// TIA Portal V15.1 export
// export: Created 2024-06-21T08:40:41.5372667Z, ExportSetting WithDefaults, DisplayName Totally Integrated Automation Portal, DisplayVersion V15.1 Update 5, DisplayName TIA Portal Openness, DisplayVersion V15.1 Update 5, DisplayName SINAMICS Startdrive Advanced, DisplayVersion V15.1, DisplayName G130, G150, S120, S150, SINAMICS MV, S210, DisplayVersion V15.1, DisplayName G110M, G120, G120C, G120D, G120P, DisplayVersion V15.1, DisplayName STEP 7 Professional, DisplayVersion V15.1 Update 5, DisplayName STEP 7 Safety, DisplayVersion V15.1, DisplayName WinCC Professional, DisplayVersion V15.1 Update 5, DisplayName SIMATIC Visualization Architect, DisplayVersion V15.1
DATA_BLOCK "_209000NCP01Passiv"   // DB252
{ S7_Optimized_Access := 'FALSE' }
AUTHOR : VCC
VERSION : 0.1
// stored: AutoNumber false, DBAccessibleFromOPCUA true, IsOnlyStoredInLoadMemory false, IsWriteProtectedInAS false
   VAR RETAIN
      AA_209000AK01JX35IF5010 { ExternalAccessible := 'False'; ExternalVisible := 'False'; ExternalWritable := 'False'} : Bool;   // Passivation alarm - ET200sp I/O - Safety Card IF5010
      AA_209000AS01JX38IF5100 { ExternalAccessible := 'False'; ExternalVisible := 'False'; ExternalWritable := 'False'} : Bool;   // Passivation alarm - ET200sp I/O - Safety Card IF5100
      AA_209000AS02JX39IF5130 { ExternalAccessible := 'False'; ExternalVisible := 'False'; ExternalWritable := 'False'} : Bool;   // Passivation alarm - ET200sp I/O - Safety Card IF5130
      AA_211212AE1JX200IF29000 { ExternalAccessible := 'False'; ExternalVisible := 'False'; ExternalWritable := 'False'} : Bool;   // Passivation alarm - ET200sp I/O - Safety Card IF29000
      AA_211212AE1JX200IF29006 { ExternalAccessible := 'False'; ExternalVisible := 'False'; ExternalWritable := 'False'} : Bool;   // Passivation alarm - ET200sp I/O - Safety Card IF29006
      AA_211212AE1JX200QF29012 { ExternalAccessible := 'False'; ExternalVisible := 'False'; ExternalWritable := 'False'} : Bool;   // Passivation alarm - ET200sp I/O - Safety Card QF29012
      AA_211212AE1JX200QF29018 { ExternalAccessible := 'False'; ExternalVisible := 'False'; ExternalWritable := 'False'} : Bool;   // Passivation alarm - ET200sp I/O - Safety Card QF29018
      "209000AK01JX35IF5010AlarmABCondition" { ExternalAccessible := 'False'; ExternalVisible := 'False'; ExternalWritable := 'False'} : Bool;   // Alarm AB condition
      "209000AS01JX38IF5100AlarmABCondition" { ExternalAccessible := 'False'; ExternalVisible := 'False'; ExternalWritable := 'False'} : Bool;   // Alarm AB condition
      "209000AS02JX39IF5130AlarmABCondition" { ExternalAccessible := 'False'; ExternalVisible := 'False'; ExternalWritable := 'False'} : Bool;   // Alarm AB condition
      "211212AE1JX200IF29000AlarmABCondition" { ExternalAccessible := 'False'; ExternalVisible := 'False'; ExternalWritable := 'False'} : Bool;   // Alarm AB condition
      "211212AE1JX200IF29006AlarmABCondition" { ExternalAccessible := 'False'; ExternalVisible := 'False'; ExternalWritable := 'False'} : Bool;   // Alarm AB condition
      "211212AE1JX200QF29012AlarmABCondition" { ExternalAccessible := 'False'; ExternalVisible := 'False'; ExternalWritable := 'False'} : Bool;   // Alarm AB condition
      "211212AE1JX200QF29018AlarmABCondition" { ExternalAccessible := 'False'; ExternalVisible := 'False'; ExternalWritable := 'False'} : Bool;   // Alarm AB condition
      H_209000AK01JX35IF5010IAnim : Word;   // HMI Animation of the icon
      H_209000AS01JX38IF5100IAnim : Word;   // HMI Animation of the icon
      H_209000AS02JX39IF5130IAnim : Word;   // HMI Animation of the icon
      H_211212AE1JX200IF29000IAnim : Word;   // HMI Animation of the icon
      H_211212AE1JX200IF29006IAnim : Word;   // HMI Animation of the icon
      H_211212AE1JX200QF29012IAnim : Word;   // HMI Animation of the icon
      H_211212AE1JX200QF29018IAnim : Word;   // HMI Animation of the icon
      H_Anim : Word;   // Animation
      H_DBnr : Int;   // DB number
      H_HMICmd : Word;   // HMI command
      AlarmA { ExternalAccessible := 'False'; ExternalVisible := 'False'; ExternalWritable := 'False'} : Bool;   // Summary Alarm A
      AlarmB { ExternalAccessible := 'False'; ExternalVisible := 'False'; ExternalWritable := 'False'} : Bool;   // Summary Alarm B
      AlarmC { ExternalAccessible := 'False'; ExternalVisible := 'False'; ExternalWritable := 'False'} : Bool;   // Summary Alarm C
      AlarmD { ExternalAccessible := 'False'; ExternalVisible := 'False'; ExternalWritable := 'False'} : Bool;   // Summary Alarm D
      AlarmABCondition { ExternalAccessible := 'False'; ExternalVisible := 'False'; ExternalWritable := 'False'} : Bool;   // Alarm AB Condition
      PassivationError { ExternalAccessible := 'False'; ExternalVisible := 'False'; ExternalWritable := 'False'} : Bool;   // There is one ore more Passivation Errors active
      FeedBackError { ExternalAccessible := 'False'; ExternalVisible := 'False'; ExternalWritable := 'False'} : Bool;   // There is one ore more FeedBack Errors active
      "AckReqSendRcvDP/PN" { ExternalAccessible := 'False'; ExternalVisible := 'False'; ExternalWritable := 'False'} : Bool;   // Ack.Req from DP/DP or PN/PN couplers
      HMIResetPassivation { ExternalAccessible := 'False'; ExternalVisible := 'False'; ExternalWritable := 'False'} : Bool;   // Reset Passivation alarm from HMI
   END_VAR
BEGIN
END_DATA_BLOCK
